// TIA Portal V19 export
FUNCTION_BLOCK "ButtonsHMIDecoder"   // FB83, LAD
// stored: Access Published, MemoryReserve 100, SetENOAutomatically false
   VAR_INPUT
      ButtonMinus : Bool;
      ButtonPlus : Bool;
      OpEnabled : Bool;
      OpRunning : Bool;
      OpDone : Bool;
      CodeReq : Int;
   END_VAR
   VAR_OUTPUT
      Code : Int;
      OperationMinus : Bool;
      OperationPlus : Bool;
      Lamp : Bool;
   END_VAR
   VAR
      SavedCode : Int;
      PE_Aux_ButtonMinus : Bool;
      PE_Aux_ButtonPlus : Bool;
      tonStable : TON_TIME;
   END_VAR
   VAR_TEMP
      CodeEqual : Bool;
   END_VAR
   VAR CONSTANT
      STABLE_TIME : Time := t#50ms;
   END_VAR
   VAR_TEMP   // added for the SCL form of the ladder/FBD networks
      _w1 : Bool;
      _w2 : Bool;
   END_VAR
BEGIN

REGION Network 1
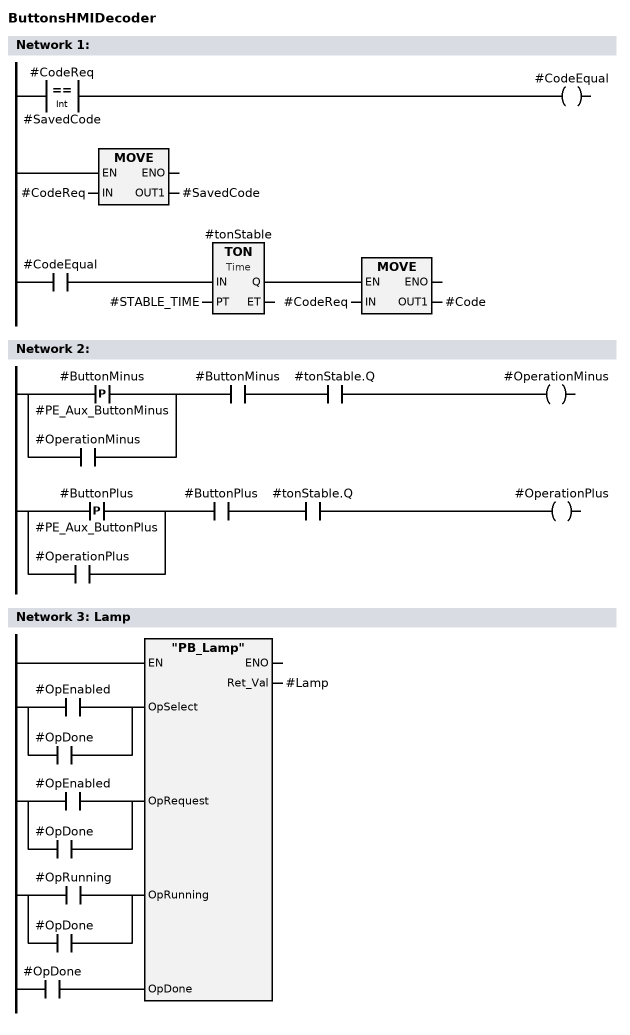
   RUNG wire#powerrail
      { S7_Templates := "SrcType := Int" } EQ_Contact(in1 := #CodeReq, in2 := #SavedCode)
      Coil( #CodeEqual )
   END_RUNG
   RUNG wire#powerrail
      Move(in := #CodeReq, out1 => #SavedCode)
   END_RUNG
   RUNG wire#powerrail
      Contact( #CodeEqual )
      { S7_Templates := "time_type := Time" } #tonStable.TON(pt := #STABLE_TIME, et =>)
      Move(in := #CodeReq, out1 => #Code)
   END_RUNG
   // the same network as SCL:
   #CodeEqual := #CodeReq = #SavedCode;
   #SavedCode := #CodeReq;
   #tonStable(IN := #CodeEqual, PT := #STABLE_TIME);   // TON
   IF #tonStable.Q THEN #Code := #CodeReq; END_IF;
END_REGION

REGION Network 2
   RUNG wire#powerrail
      P_Contact(operand := #ButtonMinus, bit := #PE_Aux_ButtonMinus)
      wire#w1
      Contact( #ButtonMinus )
      Contact( #tonStable.Q )
      Coil( #OperationMinus )
   END_RUNG
   RUNG wire#powerrail
      Contact( #OperationMinus )
   END_RUNG wire#w1
   RUNG wire#powerrail
      P_Contact(operand := #ButtonPlus, bit := #PE_Aux_ButtonPlus)
      wire#w2
      Contact( #ButtonPlus )
      Contact( #tonStable.Q )
      Coil( #OperationPlus )
   END_RUNG
   RUNG wire#powerrail
      Contact( #OperationPlus )
   END_RUNG wire#w2
   // the same network as SCL:
   #_w1 := #ButtonMinus AND NOT #PE_Aux_ButtonMinus;   // rising edge of #ButtonMinus
   #PE_Aux_ButtonMinus := #ButtonMinus;
   #OperationMinus := (#_w1 OR #OperationMinus) AND #ButtonMinus AND #tonStable.Q;
   #_w2 := #ButtonPlus AND NOT #PE_Aux_ButtonPlus;   // rising edge of #ButtonPlus
   #PE_Aux_ButtonPlus := #ButtonPlus;
   #OperationPlus := (#_w2 OR #OperationPlus) AND #ButtonPlus AND #tonStable.Q;
END_REGION

REGION Network 3: Lamp
   RUNG wire#powerrail
      "PB_Lamp"(OpSelect := wire#w1, OpRequest := wire#w2, OpRunning := wire#w3, OpDone := wire#w4, Ret_Val => #Lamp)
   END_RUNG
   RUNG wire#powerrail
      Contact( #OpEnabled )
   END_RUNG wire#w1
   RUNG wire#powerrail
      Contact( #OpDone )
   END_RUNG wire#w1
   RUNG wire#powerrail
      Contact( #OpEnabled )
   END_RUNG wire#w2
   RUNG wire#powerrail
      Contact( #OpDone )
   END_RUNG wire#w2
   RUNG wire#powerrail
      Contact( #OpRunning )
   END_RUNG wire#w3
   RUNG wire#powerrail
      Contact( #OpDone )
   END_RUNG wire#w3
   RUNG wire#powerrail
      Contact( #OpDone )
   END_RUNG wire#w4
   // the same network as SCL:
   #Lamp := "PB_Lamp"(OpSelect := #OpEnabled OR #OpDone,
                      OpRequest := #OpEnabled OR #OpDone,
                      OpRunning := #OpRunning OR #OpDone,
                      OpDone := #OpDone);
END_REGION
END_FUNCTION_BLOCK
